(* IEC 61131-3 sources: ax-factoryio-assembler/test, 2 files *)

(* ---- Assembler.st ---- *)
USING Demo.Utils;
USING Demo.ControlModule;
USING Demo.ControlModule.States.TwoAxisPickPlace;
USING AxUnit;
USING Demo.EquipmentModule;

NAMESPACE EquipmentModuleTest
    {TestFixture}
    CLASS AssemblerTest
        VAR PRIVATE
            assembler: TestAssembler;
            lidConveyor : MockConveyor;
            baseConveyor : MockConveyor;
            baseAtPlaceSensor : MockObjectSensor;
            partLeavingSensor : MockObjectSensor;
            lidAtPlaceSensor : MockObjectSensor;
            baseClamp : MockClamp;
            lidClamp : MockClamp;
            twoAxisPickPlace : MockTwoAxisPickPlace;
            counter: DINT;
            baseAtPlaceDelayTimer: MockTimer;
            lidAtPlaceDelayTimer: MockTimer;
            normalDelayTimer: MockTimer;
        END_VAR

        {TestSetup}
        METHOD PUBLIC SetUp
            baseConveyor.Setup();
            lidConveyor.Setup();
            baseAtPlaceSensor.Setup();
            lidAtPlaceSensor.Setup();
            partLeavingSensor.Setup();
            baseClamp.Setup();
            lidClamp.Setup();
            twoAxisPickPlace.Setup();
            baseAtPlaceDelayTimer.SetDuration(LTIME#1s);
            lidAtPlaceDelayTimer.SetDuration(LTIME#1s);
            normalDelayTimer.SetDuration(LTIME#1s);
            counter:=0;

            assembler.baseConveyor := baseConveyor;
            assembler.lidConveyor := lidConveyor;
            assembler.baseAtPlaceSensor := baseAtPlaceSensor;
            assembler.lidAtPlaceSensor := lidAtPlaceSensor;
            assembler.partLeavingSensor := partLeavingSensor;
            assembler.baseClamp := baseClamp;
            assembler.lidClamp := lidClamp;
            assembler.twoAxisPickPlace := twoAxisPickPlace;
            assembler.baseAtPlaceDelayTimer := baseAtPlaceDelayTimer;
            assembler.lidAtPlaceDelayTimer := lidAtPlaceDelayTimer;
            assembler.normalDelayTimer := normalDelayTimer;
            assembler.counter := REF(Counter);
            assembler.Setup();
        END_METHOD

        {Test}
        METHOD PUBLIC Should_Be_In_Idle_Status_When_Inited
            Assert.Equal(actual := assembler.GetStatus(), expected := AssemblerStatus#IDLE);
        END_METHOD

        {Test}
        METHOD PUBLIC Should_Move_To_Starting_Status_When_StartButtonPressed
            assembler.Start();

            Assert.Equal(actual := assembler.GetStatus(), expected := AssemblerStatus#STARTED);
        END_METHOD

        {Test}
        METHOD PUBLIC Should_Move_Keep_Current_status_If_Not_In_Idle_Status_When_StartButtonPressed
            assembler.SetStatus(AssemblerStatus#CLAMPING_PARTS);

            assembler.Start();

            Assert.Equal(actual := assembler.GetStatus(), expected := AssemblerStatus#CLAMPING_PARTS);
        END_METHOD

        {Test}
        METHOD PUBLIC Should_Start_Moving_Conveyors_When_Status_Is_Started
            assembler.Start();
            assembler.Cycle();

            Assert.Equal(actual := baseConveyor.started, expected := TRUE);
            Assert.Equal(actual := lidConveyor.started, expected := TRUE);
            Assert.Equal(actual := assembler.GetStatus(), expected := AssemblerStatus#WAITING_FOR_PARTS);
        END_METHOD

        {Test}
        METHOD PUBLIC Should_Stop_BaseConveyor_When_Base_Arrived
            baseConveyor.started := TRUE;
            lidConveyor.started := TRUE;
            assembler.SetStatus(AssemblerStatus#WAITING_FOR_PARTS);
            baseAtPlaceDelayTimer.timeUp :=TRUE;

            assembler.Cycle();

            Assert.Equal(actual := baseConveyor.started, expected := FALSE);
            Assert.Equal(actual := lidConveyor.started, expected := TRUE);
            Assert.Equal(actual := baseClamp.clamped, expected := TRUE);
            Assert.Equal(actual := assembler.GetStatus(), expected := AssemblerStatus#WAITING_FOR_PARTS);
        END_METHOD

        {Test}
        METHOD PUBLIC Should_Stop_Both_Conveyor_And_Clamp_Both_Parts_When_Lid_And_Base_Arrived
            baseConveyor.started := TRUE;
            lidConveyor.started := TRUE;
            assembler.SetStatus(AssemblerStatus#WAITING_FOR_PARTS);
            baseAtPlaceDelayTimer.timeUp :=TRUE;
            lidAtPlaceDelayTimer.timeUp :=TRUE;

            assembler.Cycle();

            Assert.Equal(actual := baseConveyor.started, expected := FALSE);
            Assert.Equal(actual := lidConveyor.started, expected := FALSE);
            Assert.Equal(actual := baseClamp.clamped, expected := TRUE);
            Assert.Equal(actual := lidClamp.clamped, expected := TRUE);
            Assert.Equal(actual := assembler.GetStatus(), expected := AssemblerStatus#CLAMPING_PARTS);
        END_METHOD

        {Test}
        METHOD PUBLIC Should_Release_Clamps_And_Start_AxixPickPlace_When_ClampingParts
            baseClamp.clamped := TRUE;
            lidClamp.clamped := TRUE;
            assembler.SetStatus(AssemblerStatus#CLAMPING_PARTS);
            normalDelayTimer.timeUp := TRUE;

            assembler.Cycle();

            Assert.Equal(actual := baseClamp.clamped, expected := FALSE);
            Assert.Equal(actual := lidClamp.clamped, expected := FALSE);
            Assert.Equal(actual := twoAxisPickPlace.GetIsDone(), expected := FALSE);
            Assert.Equal(actual := twoAxisPickPlace.mockState, expected := MockTwoAxisPickPlaceStatus#STARTED);
            Assert.Equal(actual := assembler.GetStatus(), expected := AssemblerStatus#PICK_AND_PLACE);
        END_METHOD
    END_CLASS
END_NAMESPACE

(* ---- Button.st ---- *)
USING AxUnit;
USING Demo.ControlModule;

NAMESPACE ControlModuleTest
    {TestFixture}
    CLASS ButtonTests
        VAR PRIVATE
            _hmi:BOOL;
            _signal:BOOL;
            _myButton: Button;
        END_VAR

        {Test(signal:=FALSE, result:=FALSE)}
        {Test(signal:=TRUE, result:=TRUE)}
        METHOD PUBLIC Button_Should_BePressed_Given_Input_Without_HMI_Signal
            VAR_INPUT
                signal: BOOL;
                result:BOOL;
            END_VAR

            _signal := signal;

            _myButton.Signal := REF(_signal);
            _myButton.HMI := NULL;
            Assert.Equal(actual := _myButton.IsPressed(), expected := result);
        END_METHOD

        {Test(signal:=FALSE, hmi:=TRUE, result:=TRUE)}
        {Test(signal:=FALSE, hmi:=FALSE, result:=FALSE)}
        {Test(signal:=TRUE, hmi:=FALSE, result:=TRUE)}
        {Test(signal:=TRUE, hmi:=TRUE, result:=TRUE)}
        METHOD PUBLIC Button_Should_BePressed_Given_Input_OR_HMI_Signal
            VAR_INPUT
                signal: BOOL;
                hmi: BOOL;
                result:BOOL;
            END_VAR
            _signal := signal;
            _hmi := hmi;

            _myButton.Signal := REF(_signal);
            _myButton.HMI := REF(_hmi);
            Assert.Equal(actual := _myButton.IsPressed(), expected := result);
        END_METHOD
    END_CLASS

    {TestFixture}
    CLASS ButtonWithLightTests
        VAR PRIVATE
            _signal:BOOL;
            _hmi: BOOL;
            _lightSignal:BOOL;
            _myButtonWithLight: ButtonWithLight;
        END_VAR

        {Test(signal:=FALSE, result:=FALSE)}
        {Test(signal:=TRUE, result:=TRUE)}
        METHOD PUBLIC Light_Should_LightUp_Given_Input_Only
            VAR_INPUT
                signal: BOOL;
                result:BOOL;
            END_VAR
            _signal := signal;

            _myButtonWithLight.Signal := REF(_signal);
            _myButtonWithLight.HMI := NULL;
            _myButtonWithLight.LightSignal := REF(_lightSignal);

            _myButtonWithLight.Cycle();

            Assert.Equal(actual := _lightSignal, expected := result);
        END_METHOD

        {Test(signal:=FALSE, hmi:=TRUE, result:=FALSE)}
        {Test(signal:=TRUE, hmi:=FALSE, result:=TRUE)}
        METHOD PUBLIC Light_Should_LightUp_According_To_Input_Not_HMI
            VAR_INPUT
                signal: BOOL;
                result:BOOL;
                hmi:BOOL;
            END_VAR
            _signal := signal;
            _hmi := hmi;

            _myButtonWithLight.Signal := REF(_signal);
            _myButtonWithLight.HMI := REF(_hmi);
            _myButtonWithLight.LightSignal := REF(_lightSignal);

            _myButtonWithLight.Cycle();

            Assert.Equal(actual := _lightSignal, expected := result);
        END_METHOD
    END_CLASS

END_NAMESPACE
